Yaskawa INFORM job: 5.JBI

/JOB
//NAME 5
//POS
///NPOS 6,0,0,0
///TOOL 0
///PULSE
C000=-11160,36781,-37557,130,7785,3489
C001=-9365,43572,-35071,2383,7025,1960
C002=-12888,32495,-38253,-7513,7588,8473
C003=-10444,29801,-38327,-7544,8177,8336
C004=-13078,33440,-40090,-11897,7367,11294
C005=-13078,32579,-29295,-1001,5577,4266
//INST
///DATE 2014/10/13 01:02
///ATTR 0,0,0,0,0,0,0,0,0,0,0,0,0,1,0,0
///FRAME BASE
NOP
MOVJ C000 VJ=0.78 CONT
MOVJ C001 VJ=0.78 CONT
MOVJ C002 VJ=0.78 CONT
MOVJ C003 VJ=0.78 CONT
MOVJ C004 VJ=0.78 CONT
MOVJ C005 VJ=0.78 CONT
END
